PROGRAM TimeTrackerCtrl
VAR
	tTrackerResetDelay			: ARRAY[0..iProductRecipeArrayQty] OF TON;

	fbV2MinMaxExtShift			: fbV2_MinMaxExtShift;

END_VAR
VAR // added by the converter: edge detectors and wires of the graphical bodies
    _w1 : INT;
END_VAR

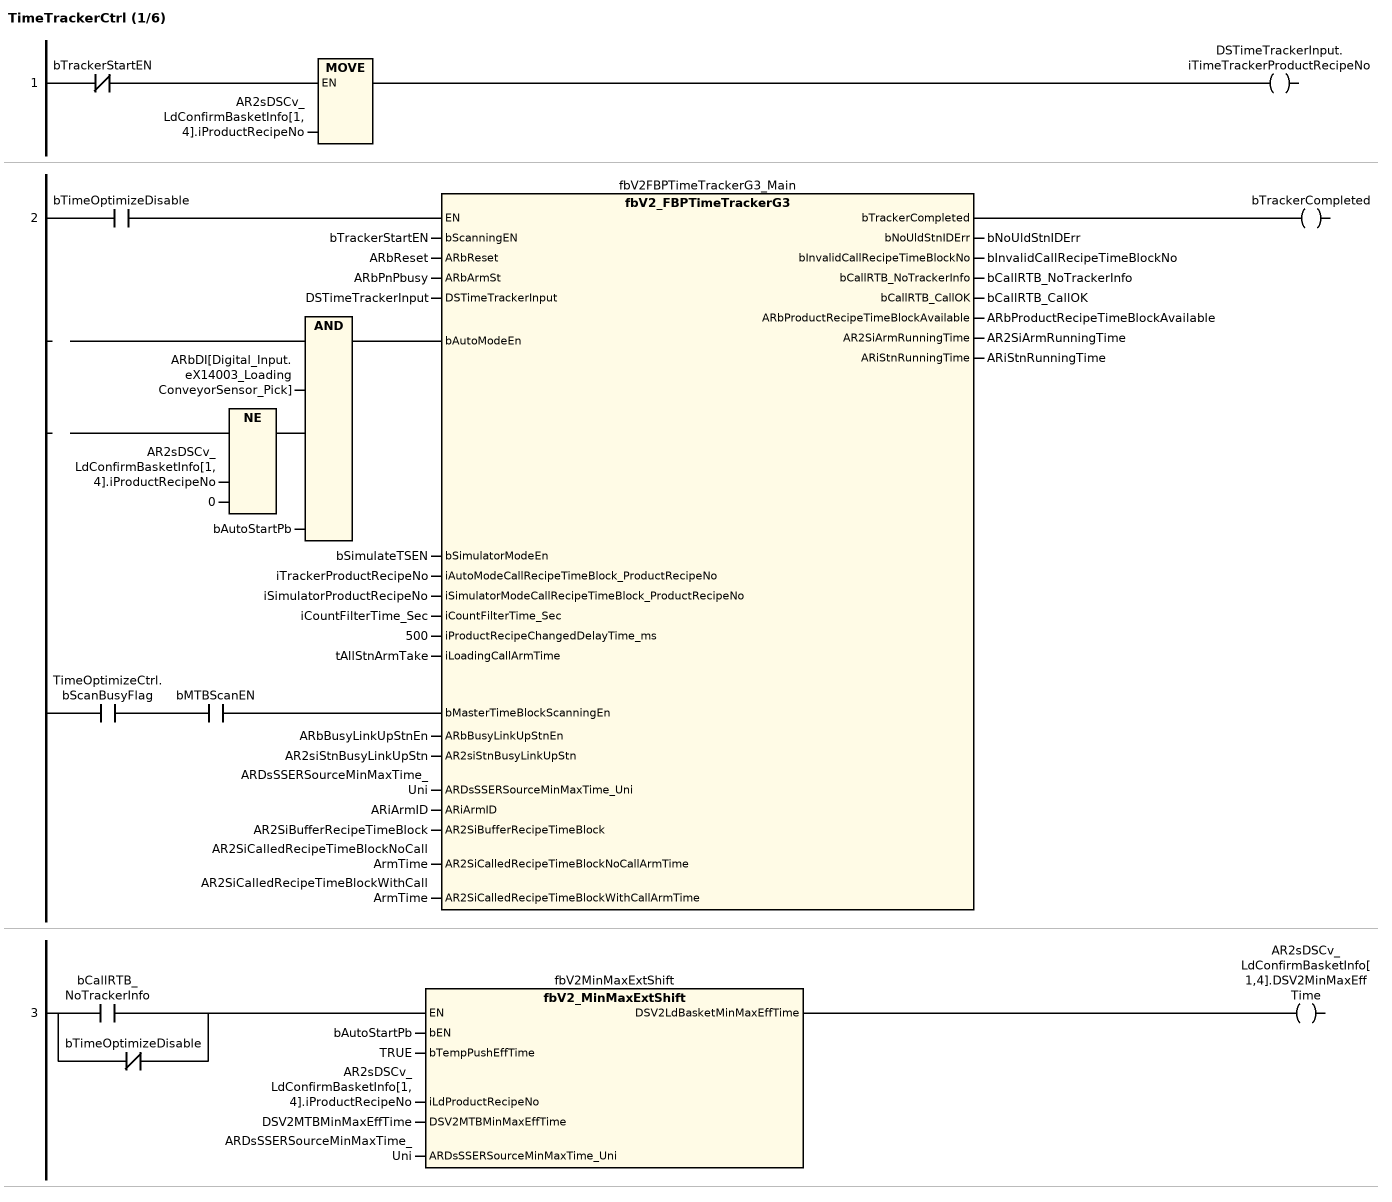
// NETWORK 1
IF NOT bTrackerStartEN THEN _w1 := AR2sDSCv_LdConfirmBasketInfo[1,4].iProductRecipeNo; END_IF
DSTimeTrackerInput.iTimeTrackerProductRecipeNo := _w1;

// NETWORK 2
IF bTimeOptimizeDisable THEN
    fbV2FBPTimeTrackerG3_Main(
        bScanningEN := bTrackerStartEN,
        ARbReset := ARbReset,
        ARbArmSt := ARbPnPbusy,
        DSTimeTrackerInput := DSTimeTrackerInput,
        bAutoModeEn := ARbDI[Digital_Input.eX14003_LoadingConveyorSensor_Pick] AND AR2sDSCv_LdConfirmBasketInfo[1,4].iProductRecipeNo <> 0 AND bAutoStartPb,
        bSimulatorModeEn := bSimulateTSEN,
        iAutoModeCallRecipeTimeBlock_ProductRecipeNo := iTrackerProductRecipeNo,
        iSimulatorModeCallRecipeTimeBlock_ProductRecipeNo := iSimulatorProductRecipeNo,
        iCountFilterTime_Sec := iCountFilterTime_Sec,
        iProductRecipeChangedDelayTime_ms := 500,
        iLoadingCallArmTime := tAllStnArmTake,
        bMasterTimeBlockScanningEn := TimeOptimizeCtrl.bScanBusyFlag AND bMTBScanEN,
        ARbBusyLinkUpStnEn := ARbBusyLinkUpStnEn,
        AR2siStnBusyLinkUpStn := AR2siStnBusyLinkUpStn,
        ARDsSSERSourceMinMaxTime_Uni := ARDsSSERSourceMinMaxTime_Uni,
        ARiArmID := ARiArmID,
        AR2SiBufferRecipeTimeBlock := AR2SiBufferRecipeTimeBlock,
        AR2SiCalledRecipeTimeBlockNoCallArmTime := AR2SiCalledRecipeTimeBlockNoCallArmTime,
        AR2SiCalledRecipeTimeBlockWithCallArmTime := AR2SiCalledRecipeTimeBlockWithCallArmTime,
        bNoUldStnIDErr => bNoUldStnIDErr,
        bInvalidCallRecipeTimeBlockNo => bInvalidCallRecipeTimeBlockNo,
        bCallRTB_NoTrackerInfo => bCallRTB_NoTrackerInfo,
        bCallRTB_CallOK => bCallRTB_CallOK,
        ARbProductRecipeTimeBlockAvailable => ARbProductRecipeTimeBlockAvailable,
        AR2SiArmRunningTime => AR2SiArmRunningTime,
        ARiStnRunningTime => ARiStnRunningTime); // fbV2_FBPTimeTrackerG3
END_IF
bTrackerCompleted := fbV2FBPTimeTrackerG3_Main.bTrackerCompleted;

// NETWORK 3
IF bCallRTB_NoTrackerInfo OR NOT bTimeOptimizeDisable THEN
    fbV2MinMaxExtShift(
        bEN := bAutoStartPb,
        bTempPushEffTime := TRUE,
        iLdProductRecipeNo := AR2sDSCv_LdConfirmBasketInfo[1,4].iProductRecipeNo,
        DSV2MTBMinMaxEffTime := DSV2MTBMinMaxEffTime,
        ARDsSSERSourceMinMaxTime_Uni := ARDsSSERSourceMinMaxTime_Uni); // fbV2_MinMaxExtShift
END_IF
AR2sDSCv_LdConfirmBasketInfo[1,4].DSV2MinMaxEffTime := fbV2MinMaxExtShift.DSV2LdBasketMinMaxEffTime;

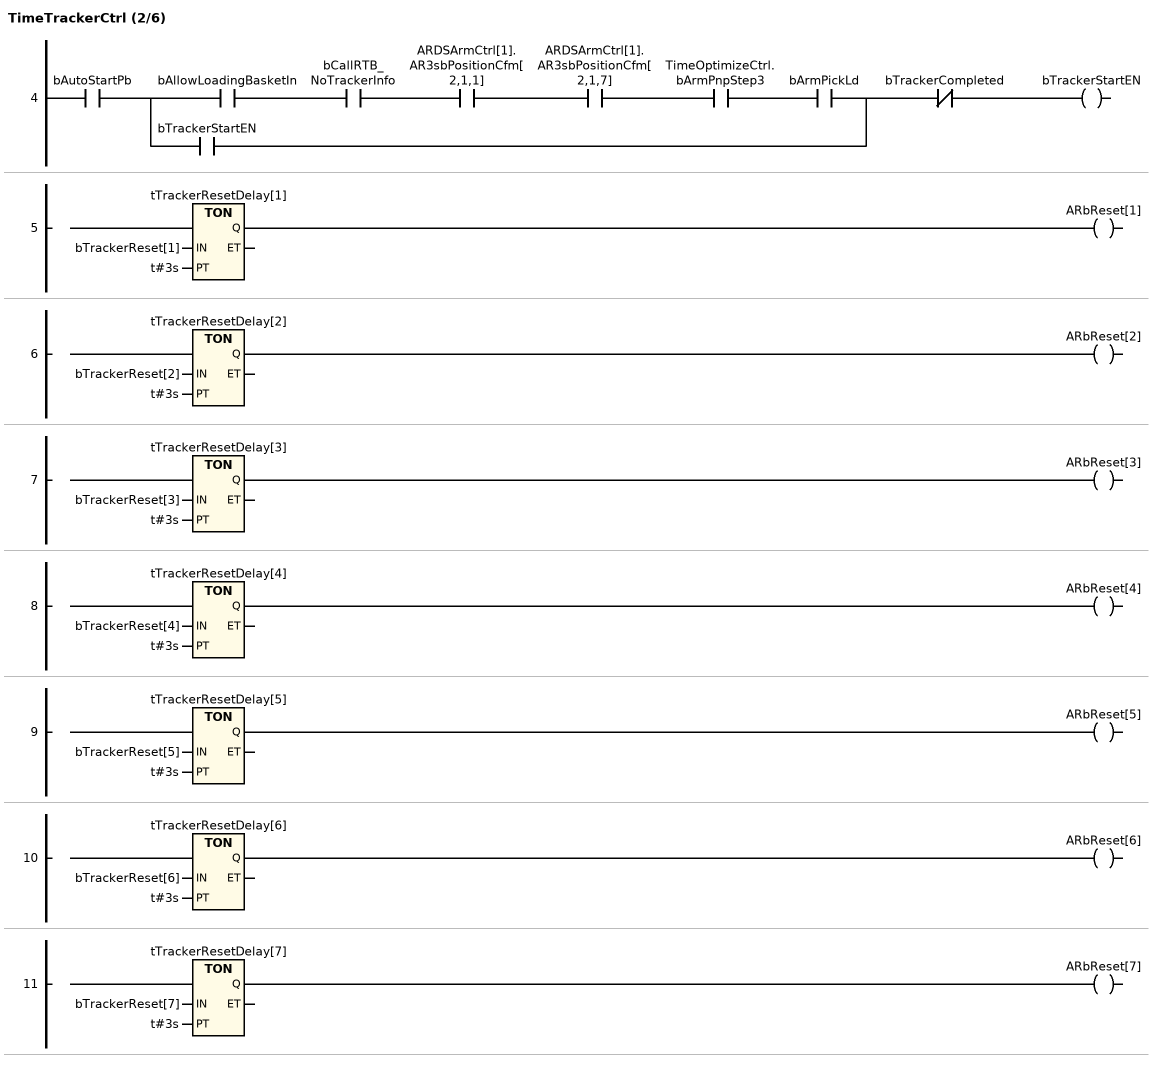
// NETWORK 4
bTrackerStartEN := (bAutoStartPb AND (bAllowLoadingBasketIn AND bCallRTB_NoTrackerInfo AND ARDSArmCtrl[1].AR3sbPositionCfm[2,1,1] AND ARDSArmCtrl[1].AR3sbPositionCfm[2,1,7] AND TimeOptimizeCtrl.bArmPnpStep3 AND bArmPickLd OR bTrackerStartEN)) AND NOT bTrackerCompleted;

// NETWORK 5
tTrackerResetDelay[1](IN := bTrackerReset[1], PT := t#3s); // TON
ARbReset[1] := tTrackerResetDelay[1].Q;

// NETWORK 6
tTrackerResetDelay[2](IN := bTrackerReset[2], PT := t#3s); // TON
ARbReset[2] := tTrackerResetDelay[2].Q;

// NETWORK 7
tTrackerResetDelay[3](IN := bTrackerReset[3], PT := t#3s); // TON
ARbReset[3] := tTrackerResetDelay[3].Q;

// NETWORK 8
tTrackerResetDelay[4](IN := bTrackerReset[4], PT := t#3s); // TON
ARbReset[4] := tTrackerResetDelay[4].Q;

// NETWORK 9
tTrackerResetDelay[5](IN := bTrackerReset[5], PT := t#3s); // TON
ARbReset[5] := tTrackerResetDelay[5].Q;

// NETWORK 10
tTrackerResetDelay[6](IN := bTrackerReset[6], PT := t#3s); // TON
ARbReset[6] := tTrackerResetDelay[6].Q;

// NETWORK 11
tTrackerResetDelay[7](IN := bTrackerReset[7], PT := t#3s); // TON
ARbReset[7] := tTrackerResetDelay[7].Q;

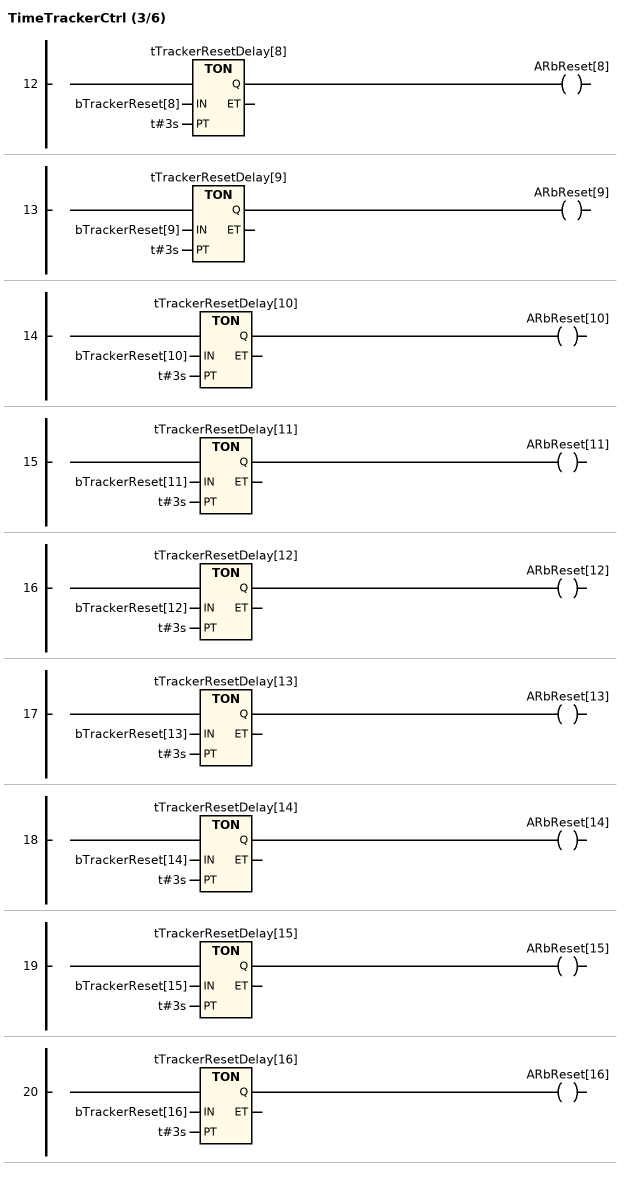
// NETWORK 12
tTrackerResetDelay[8](IN := bTrackerReset[8], PT := t#3s); // TON
ARbReset[8] := tTrackerResetDelay[8].Q;

// NETWORK 13
tTrackerResetDelay[9](IN := bTrackerReset[9], PT := t#3s); // TON
ARbReset[9] := tTrackerResetDelay[9].Q;

// NETWORK 14
tTrackerResetDelay[10](IN := bTrackerReset[10], PT := t#3s); // TON
ARbReset[10] := tTrackerResetDelay[10].Q;

// NETWORK 15
tTrackerResetDelay[11](IN := bTrackerReset[11], PT := t#3s); // TON
ARbReset[11] := tTrackerResetDelay[11].Q;

// NETWORK 16
tTrackerResetDelay[12](IN := bTrackerReset[12], PT := t#3s); // TON
ARbReset[12] := tTrackerResetDelay[12].Q;

// NETWORK 17
tTrackerResetDelay[13](IN := bTrackerReset[13], PT := t#3s); // TON
ARbReset[13] := tTrackerResetDelay[13].Q;

// NETWORK 18
tTrackerResetDelay[14](IN := bTrackerReset[14], PT := t#3s); // TON
ARbReset[14] := tTrackerResetDelay[14].Q;

// NETWORK 19
tTrackerResetDelay[15](IN := bTrackerReset[15], PT := t#3s); // TON
ARbReset[15] := tTrackerResetDelay[15].Q;

// NETWORK 20
tTrackerResetDelay[16](IN := bTrackerReset[16], PT := t#3s); // TON
ARbReset[16] := tTrackerResetDelay[16].Q;

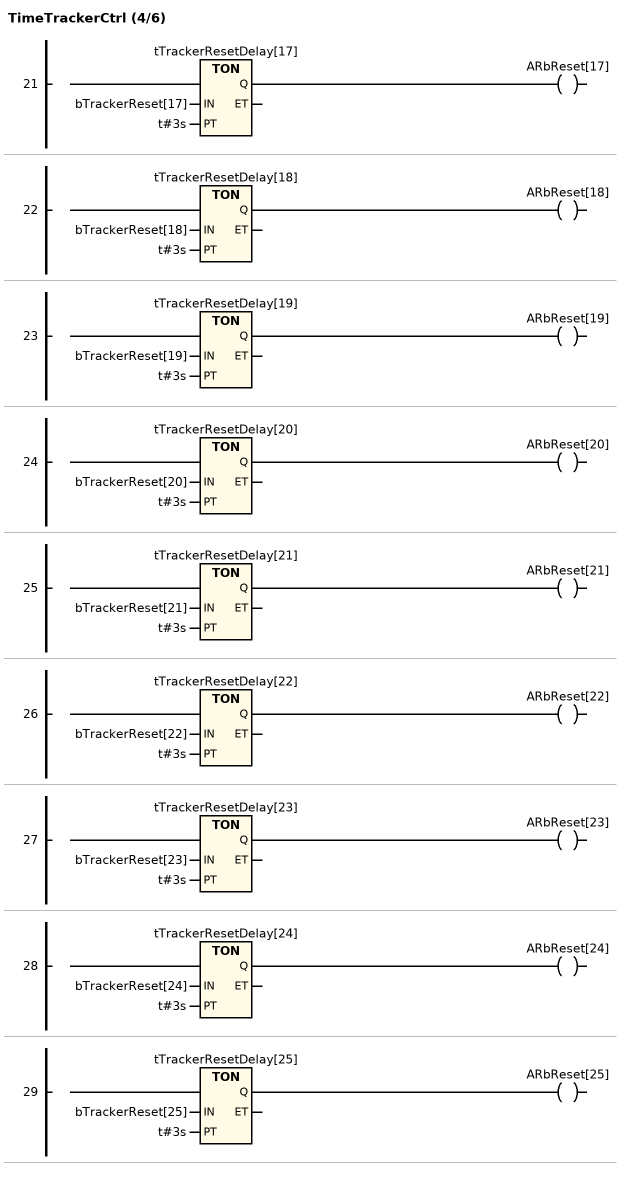
// NETWORK 21
tTrackerResetDelay[17](IN := bTrackerReset[17], PT := t#3s); // TON
ARbReset[17] := tTrackerResetDelay[17].Q;

// NETWORK 22
tTrackerResetDelay[18](IN := bTrackerReset[18], PT := t#3s); // TON
ARbReset[18] := tTrackerResetDelay[18].Q;

// NETWORK 23
tTrackerResetDelay[19](IN := bTrackerReset[19], PT := t#3s); // TON
ARbReset[19] := tTrackerResetDelay[19].Q;

// NETWORK 24
tTrackerResetDelay[20](IN := bTrackerReset[20], PT := t#3s); // TON
ARbReset[20] := tTrackerResetDelay[20].Q;

// NETWORK 25
tTrackerResetDelay[21](IN := bTrackerReset[21], PT := t#3s); // TON
ARbReset[21] := tTrackerResetDelay[21].Q;

// NETWORK 26
tTrackerResetDelay[22](IN := bTrackerReset[22], PT := t#3s); // TON
ARbReset[22] := tTrackerResetDelay[22].Q;

// NETWORK 27
tTrackerResetDelay[23](IN := bTrackerReset[23], PT := t#3s); // TON
ARbReset[23] := tTrackerResetDelay[23].Q;

// NETWORK 28
tTrackerResetDelay[24](IN := bTrackerReset[24], PT := t#3s); // TON
ARbReset[24] := tTrackerResetDelay[24].Q;

// NETWORK 29
tTrackerResetDelay[25](IN := bTrackerReset[25], PT := t#3s); // TON
ARbReset[25] := tTrackerResetDelay[25].Q;

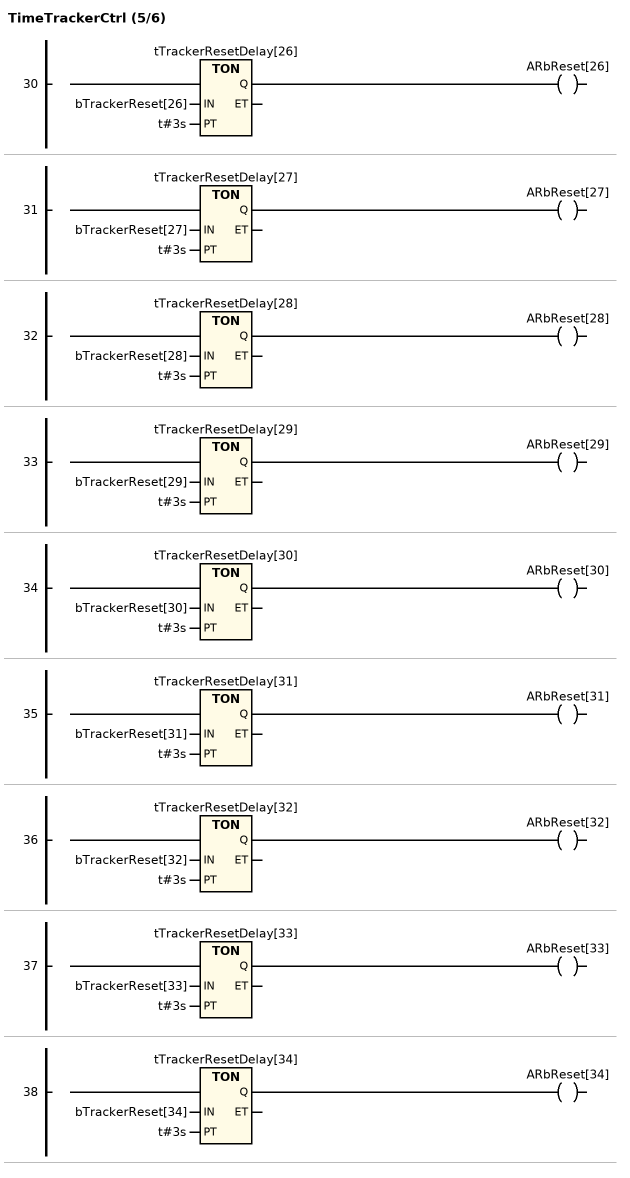
// NETWORK 30
tTrackerResetDelay[26](IN := bTrackerReset[26], PT := t#3s); // TON
ARbReset[26] := tTrackerResetDelay[26].Q;

// NETWORK 31
tTrackerResetDelay[27](IN := bTrackerReset[27], PT := t#3s); // TON
ARbReset[27] := tTrackerResetDelay[27].Q;

// NETWORK 32
tTrackerResetDelay[28](IN := bTrackerReset[28], PT := t#3s); // TON
ARbReset[28] := tTrackerResetDelay[28].Q;

// NETWORK 33
tTrackerResetDelay[29](IN := bTrackerReset[29], PT := t#3s); // TON
ARbReset[29] := tTrackerResetDelay[29].Q;

// NETWORK 34
tTrackerResetDelay[30](IN := bTrackerReset[30], PT := t#3s); // TON
ARbReset[30] := tTrackerResetDelay[30].Q;

// NETWORK 35
tTrackerResetDelay[31](IN := bTrackerReset[31], PT := t#3s); // TON
ARbReset[31] := tTrackerResetDelay[31].Q;

// NETWORK 36
tTrackerResetDelay[32](IN := bTrackerReset[32], PT := t#3s); // TON
ARbReset[32] := tTrackerResetDelay[32].Q;

// NETWORK 37
tTrackerResetDelay[33](IN := bTrackerReset[33], PT := t#3s); // TON
ARbReset[33] := tTrackerResetDelay[33].Q;

// NETWORK 38
tTrackerResetDelay[34](IN := bTrackerReset[34], PT := t#3s); // TON
ARbReset[34] := tTrackerResetDelay[34].Q;

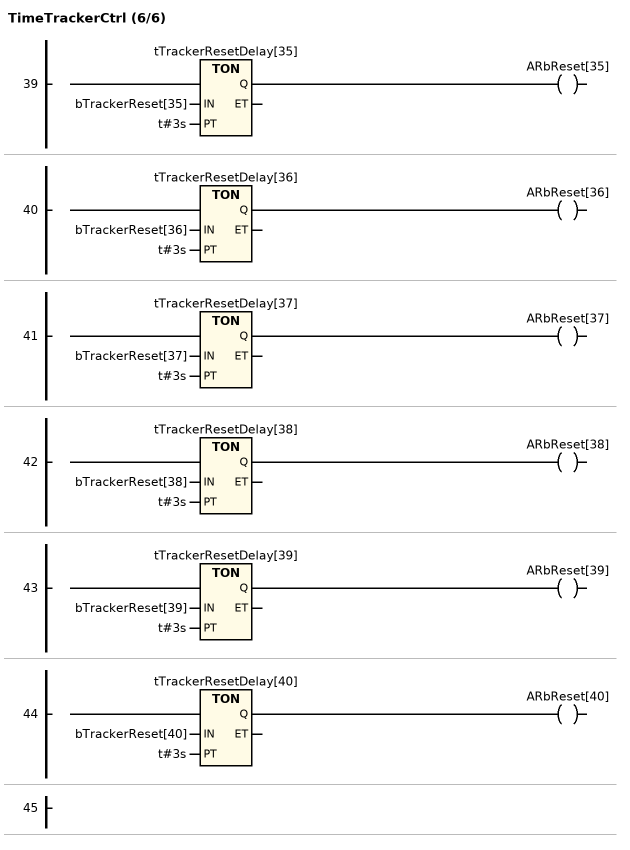
// NETWORK 39
tTrackerResetDelay[35](IN := bTrackerReset[35], PT := t#3s); // TON
ARbReset[35] := tTrackerResetDelay[35].Q;

// NETWORK 40
tTrackerResetDelay[36](IN := bTrackerReset[36], PT := t#3s); // TON
ARbReset[36] := tTrackerResetDelay[36].Q;

// NETWORK 41
tTrackerResetDelay[37](IN := bTrackerReset[37], PT := t#3s); // TON
ARbReset[37] := tTrackerResetDelay[37].Q;

// NETWORK 42
tTrackerResetDelay[38](IN := bTrackerReset[38], PT := t#3s); // TON
ARbReset[38] := tTrackerResetDelay[38].Q;

// NETWORK 43
tTrackerResetDelay[39](IN := bTrackerReset[39], PT := t#3s); // TON
ARbReset[39] := tTrackerResetDelay[39].Q;

// NETWORK 44
tTrackerResetDelay[40](IN := bTrackerReset[40], PT := t#3s); // TON
ARbReset[40] := tTrackerResetDelay[40].Q;

// NETWORK 45

END_PROGRAM

(* stored: Version 1.1.0.1, ProductVersion 3.1.4024.12
   POU TimeTrackerCtrl: Id {30711240-d5e3-47f8-9515-8f14b677cdb3}, SpecialFunc None *)
